(*
	Default Lamp device
*)
FUNCTION_BLOCK FB_Lamp EXTENDS FB_LinkDevice 
VAR_INPUT
	bEnable		: BOOL; //0-Lamp OFF, 1 - Lamp ON
END_VAR

SUPER^();
Control.0 := bEnable;

END_FUNCTION_BLOCK

(* stored: Version 1.1.0.1, ProductVersion 3.1.4024.12
   POU FB_Lamp: Id {7fc594db-b88a-0a4e-01f1-22815165cbed}, SpecialFunc None *)
